(* Logix 5000 project; controller PLC2_Project9_DDEMessaging Emulate 5570 rev 20.11; software revision 20.00 *)

TASK MainTask (continuous, watchdog 500 ms) : MainProgram

MODULES
   Local : Emulate 5570 (ICP 1, rev 20.11)
END_MODULES

PROGRAM MainProgram   (* main routine _00_Main *)
VAR
   Function : DINT; {access Read Only}   // 0: Function 1 1: Function 2
   Function_1_Timer : TIMER := (PRE := 1000); {access Read Only}
   Function_2_Timer : TIMER := (PRE := 1000); {access Read Only}
   M1F1_Cycles : DINT; {access Read Only}
   M1F2_Cycles : DINT; {access Read Only}
   M2F1_Cycles : DINT; {access Read Only}
   M2F2_Cycles : DINT; {access Read Only}
   Mode : DINT; {access Read Only}   // 0: Mode 1 1: Mode 2
   ONS_M1F1 : BOOL; {access Read Only}
   ONS_M1F2 : BOOL; {access Read Only}
   ONS_M2F1 : BOOL; {access Read Only}
   ONS_M2F2 : BOOL; {access Read Only}
   S_Function : STRING; {access Read Only}
   S_Mode : STRING; {access Read Only}
   S_ModeFunction : STRING; {access Read Only}
   TempInts : DINT[10]; {access Read Only}
   Temps : STRING[10] := ([2] := 'Function ', [3] := 'Mode '); {access Read Only}
END_VAR

ROUTINE _00_Main   (* ladder *)
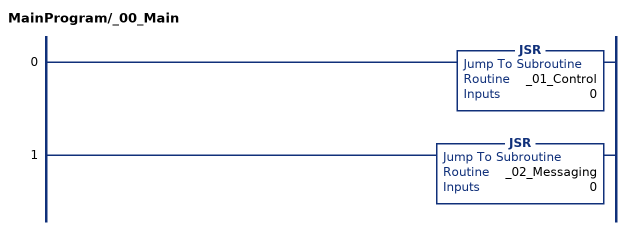
   0: JSR(_01_Control,0);
   1: JSR(_02_Messaging,0);
END_ROUTINE

ROUTINE _01_Control   (* ladder *)
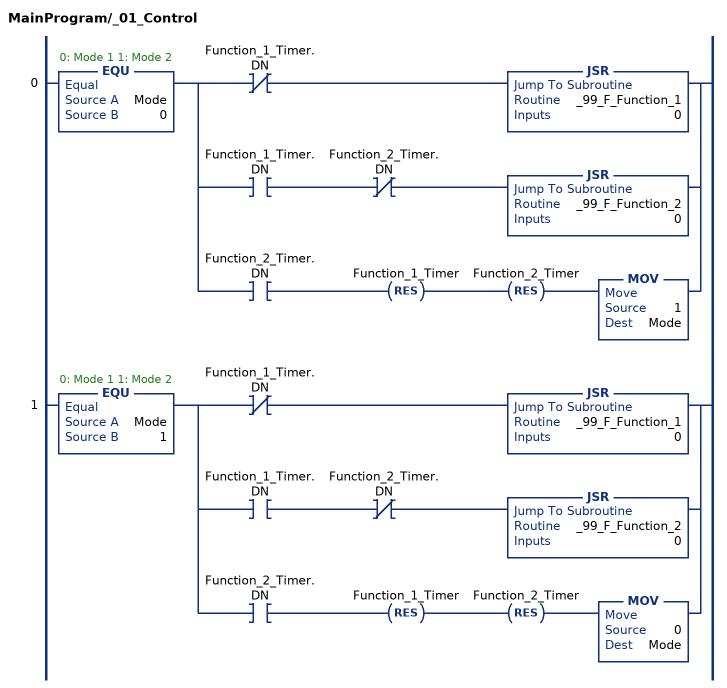
   0: EQU(Mode,0)[XIO(Function_1_Timer.DN) JSR(_99_F_Function_1,0) ,XIC(Function_1_Timer.DN) XIO(Function_2_Timer.DN) JSR(_99_F_Function_2,0) ,XIC(Function_2_Timer.DN) RES(Function_1_Timer) RES(Function_2_Timer) MOV(1,Mode) ];
   1: EQU(Mode,1)[XIO(Function_1_Timer.DN) JSR(_99_F_Function_1,0) ,XIC(Function_1_Timer.DN) XIO(Function_2_Timer.DN) JSR(_99_F_Function_2,0) ,XIC(Function_2_Timer.DN) RES(Function_1_Timer) RES(Function_2_Timer) MOV(0,Mode) ];
END_ROUTINE

ROUTINE _02_Messaging   (* ladder *)
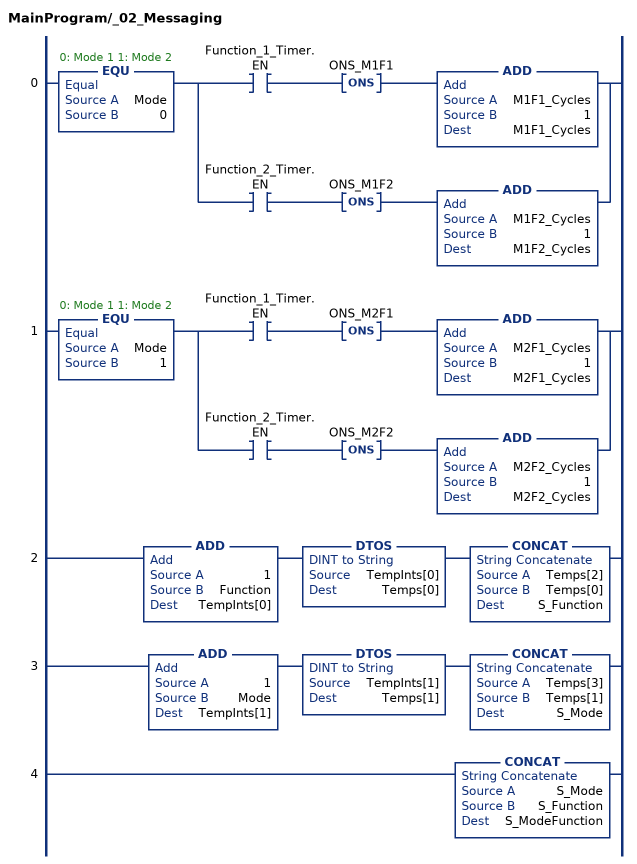
   0: EQU(Mode,0)[XIC(Function_1_Timer.EN) ONS(ONS_M1F1) ADD(M1F1_Cycles,1,M1F1_Cycles) ,XIC(Function_2_Timer.EN) ONS(ONS_M1F2) ADD(M1F2_Cycles,1,M1F2_Cycles) ];
   1: EQU(Mode,1)[XIC(Function_1_Timer.EN) ONS(ONS_M2F1) ADD(M2F1_Cycles,1,M2F1_Cycles) ,XIC(Function_2_Timer.EN) ONS(ONS_M2F2) ADD(M2F2_Cycles,1,M2F2_Cycles) ];
   2: ADD(1,Function,TempInts[0])DTOS(TempInts[0],Temps[0])CONCAT(Temps[2],Temps[0],S_Function);
   3: ADD(1,Mode,TempInts[1])DTOS(TempInts[1],Temps[1])CONCAT(Temps[3],Temps[1],S_Mode);
   4: CONCAT(S_Mode,S_Function,S_ModeFunction);
END_ROUTINE

ROUTINE _99_F_Function_1   (* ladder *)
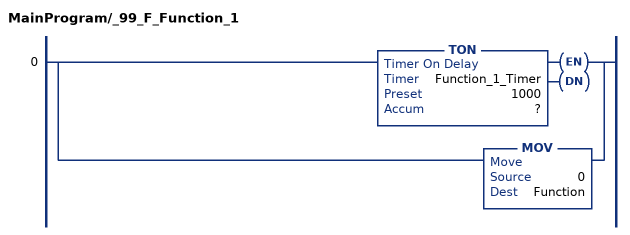
   0: [TON(Function_1_Timer,?,?) ,MOV(0,Function) ];
END_ROUTINE

ROUTINE _99_F_Function_2   (* ladder *)
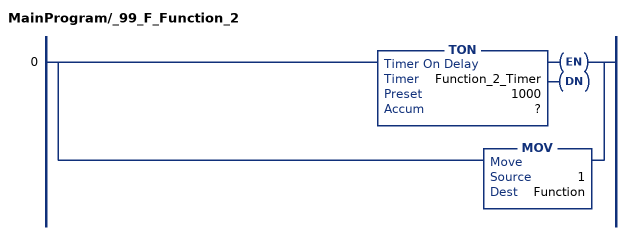
   0: [TON(Function_2_Timer,?,?) ,MOV(1,Function) ];
END_ROUTINE
END_PROGRAM
